{attribute 'enable_dynamic_creation'}
FUNCTION_BLOCK Mover IMPLEMENTS ITF_Cyclic, ITF_Mover
VAR
	myMaxVelo : LREAL;
END_VAR

{warning 'add method implementation '}
METHOD Cycle : BOOL
END_METHOD

METHOD MaxVelo : BOOL
VAR_INPUT
	MaxVelocity : LREAL;
END_VAR
END_METHOD

END_FUNCTION_BLOCK

(* stored: Version 1.1.0.1, ProductVersion 3.1.4024.12
   POU Mover: Id {5bd059eb-f1f0-4601-a642-acba93ef29cd}, SpecialFunc None
   Method Cycle: Id {7f2a9182-cb07-43c8-be8a-bfdb4121e6df}
   Method MaxVelo: Id {c3aef0a4-5c00-4d00-8076-ae1edf60ff9a} *)
